// TIA Portal V18 export
// export: Created 2025-12-01T12:38:35.135372Z, ExportSetting None, DisplayName Totally Integrated Automation Portal, DisplayVersion V18 Update 5, DisplayName TIA Portal Openness, DisplayVersion V18 Update 5, DisplayName TIA Portal Teamcenter Gateway, DisplayVersion V18, DisplayName TIA Portal Version Control Interface, DisplayVersion V18, DisplayName STEP 7 Professional, DisplayVersion V18 Update 5, DisplayName STEP 7 Safety, DisplayVersion V18, DisplayName WinCC Professional, DisplayVersion V18 Update 5
DATA_BLOCK "ST10_SafetyGate_InterfaceDB"   // DB1140
{ S7_Optimized_Access := 'TRUE' }
// stored: AutoNumber false, MemoryReserve 100
   VAR
      aDev { S7_SetPoint := 'True'} : Array[1..20] of "SafetyGateUDT";
      SafetyDoorLamp { S7_SetPoint := 'True'} : Array[1..20] of Bool;
      H : Struct
         Status_1 : Int;
         Status_2 : Int;
         Status_3 : Int;
         p : Array[0..20] of Bool;
      END_STRUCT;
      J : Struct
         Status_1 : Int;
         Status_2 : Int;
         Status_3 : Int;
         p : Array[0..20] of Bool;
      END_STRUCT;
      K : Struct
         Status_1 : Int;
         Status_2 : Int;
         Status_3 : Int;
         p : Array[0..20] of Bool;
      END_STRUCT;
      L : Struct
         Status_1 : Int;
         Status_2 : Int;
         Status_3 : Int;
         p : Array[0..20] of Bool;
      END_STRUCT;
   END_VAR
BEGIN
END_DATA_BLOCK
